TYPE ST_Chamber1DoorOpenParam :
STRUCT
END_STRUCT
END_TYPE

(* stored: Version 1.1.0.1, ProductVersion 3.1.4026.18
   DUT ST_Chamber1DoorOpenParam: Id {c3551c86-be1a-4bc3-8a57-526750a03789} *)
